// TIA Portal V17 export
// export: Created 2023-08-29T18:06:39.3261683Z, ExportSetting WithDefaults, DisplayName Totally Integrated Automation Portal, DisplayVersion V17 Update 5, DisplayName TIA Portal Openness, DisplayVersion V17 Update 5, DisplayName TIA Portal Teamcenter Gateway, DisplayVersion V17 Update 5, DisplayName TIA Portal Version Control Interface, DisplayVersion V17, DisplayName Simotion SCOUT TIA, DisplayVersion 5.4.3.0, DisplayName TIA Portal Test Suite Advanced, DisplayVersion V17 Update 1, DisplayName SIMOCODE ES, DisplayVersion V17 Update 5, DisplayName SINAMICS Startdrive Advanced, DisplayVersion V17 SP1, DisplayName SINAMICS Startdrive G130, G150, S120, S150, SINAMICS MV, S210, DisplayVersion V17 SP1, DisplayName SINAMICS Startdrive G110M, G120, G120C, G120D, G120P, G115D, DisplayVersion V17 SP1, DisplayName SIRIUS Safety ES, DisplayVersion V17 Update 5, DisplayName STEP 7 Professional, DisplayVersion V17 Update 5, DisplayName STEP 7 CFC, DisplayVersion V17 Update 1, DisplayName STEP 7 Safety, DisplayVersion V17, DisplayName WinCC Advanced, DisplayVersion V17 Update 5, DisplayName SIMATIC Visualization Architect, DisplayVersion V17 Update 5
FUNCTION "04_ESTOP" : Void   // FC5, F_FBD
TITLE = EMERGENCY STOP
{ S7_Optimized_Access := 'TRUE' }
VERSION : 0.1
// stored: AutoNumber true, IsIECCheckEnabled false, UDAEnableTagReadback false
BEGIN

REGION Network 1: !!COLUMN_1$$
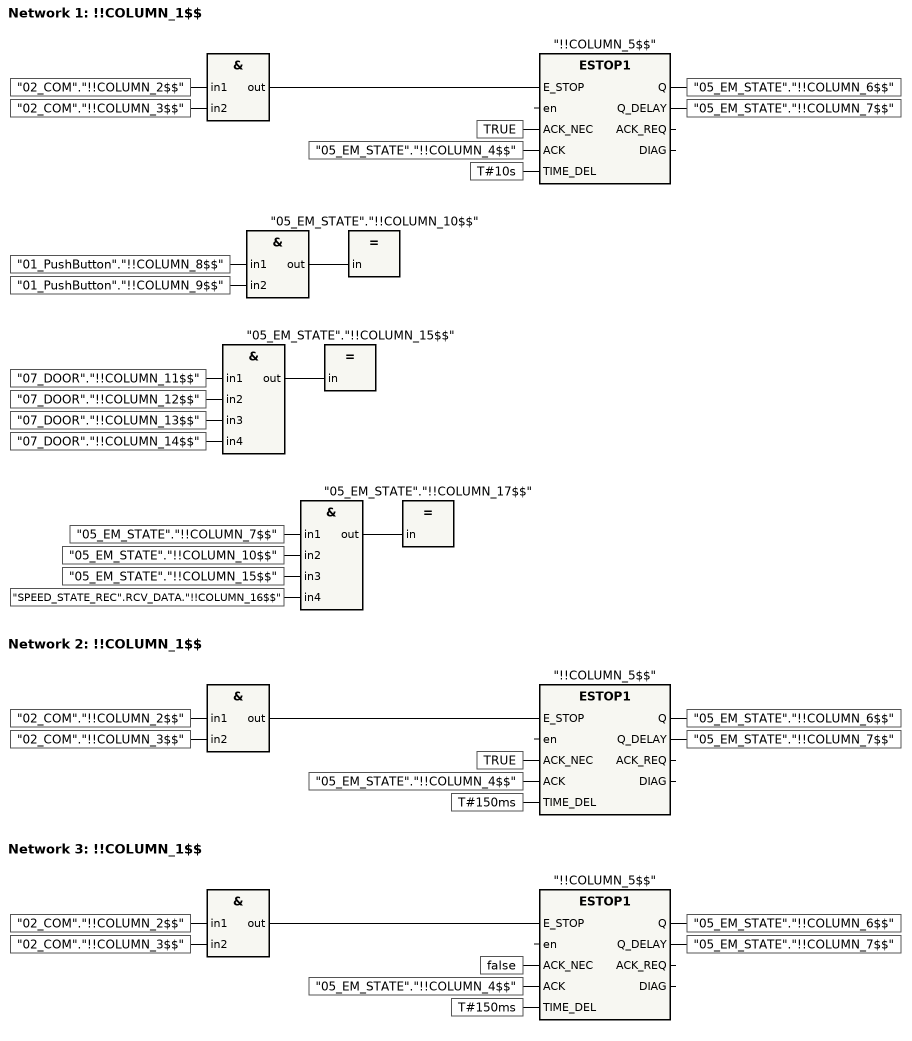
   "!!COLUMN_5$$"(E_STOP := "02_COM"."!!COLUMN_2$$" AND "02_COM"."!!COLUMN_3$$",   // ESTOP1
                  ACK_NEC := TRUE,
                  ACK := "05_EM_STATE"."!!COLUMN_4$$",
                  TIME_DEL := T#10s,
                  Q => "05_EM_STATE"."!!COLUMN_6$$",
                  Q_DELAY => "05_EM_STATE"."!!COLUMN_7$$");
   "05_EM_STATE"."!!COLUMN_10$$" := "01_PushButton"."!!COLUMN_8$$" AND "01_PushButton"."!!COLUMN_9$$";
   "05_EM_STATE"."!!COLUMN_15$$" := "07_DOOR"."!!COLUMN_11$$" AND "07_DOOR"."!!COLUMN_12$$" AND "07_DOOR"."!!COLUMN_13$$" AND "07_DOOR"."!!COLUMN_14$$";
   "05_EM_STATE"."!!COLUMN_17$$" := "05_EM_STATE"."!!COLUMN_7$$" AND "05_EM_STATE"."!!COLUMN_10$$" AND "05_EM_STATE"."!!COLUMN_15$$" AND "SPEED_STATE_REC".RCV_DATA."!!COLUMN_16$$";
END_REGION

REGION Network 2: !!COLUMN_1$$
   "!!COLUMN_5$$"(E_STOP := "02_COM"."!!COLUMN_2$$" AND "02_COM"."!!COLUMN_3$$",   // ESTOP1
                  ACK_NEC := TRUE,
                  ACK := "05_EM_STATE"."!!COLUMN_4$$",
                  TIME_DEL := T#150ms,
                  Q => "05_EM_STATE"."!!COLUMN_6$$",
                  Q_DELAY => "05_EM_STATE"."!!COLUMN_7$$");
END_REGION

REGION Network 3: !!COLUMN_1$$
   "!!COLUMN_5$$"(E_STOP := "02_COM"."!!COLUMN_2$$" AND "02_COM"."!!COLUMN_3$$",   // ESTOP1
                  ACK_NEC := false,
                  ACK := "05_EM_STATE"."!!COLUMN_4$$",
                  TIME_DEL := T#150ms,
                  Q => "05_EM_STATE"."!!COLUMN_6$$",
                  Q_DELAY => "05_EM_STATE"."!!COLUMN_7$$");
END_REGION
END_FUNCTION
